TYPE AX5000_S_0163 :
STRUCT
	Weight_counterbalance:INT;
END_STRUCT
END_TYPE

(* stored: Version 1.1.0.1, ProductVersion 3.1.4024.3
   DUT AX5000_S_0163: Id {d468a53d-b7ff-44f6-a189-2aebb02be1b6} *)
